{attribute 'GeneratedUsingTerminal: KL1382'}
{attribute addProperty BoxType "KL1382"}
{attribute addProperty Description ""}
{attribute addProperty Physics ""}
{attribute addProperty Id "Channel_1AT %I*Channel_22DCD6950Channel_2AT %I*Channel_22DCD6950"}
{attribute addProperty CRC "3041576269"}
{attribute addProperty Size "0"}
TYPE KL1382_B54AC54D :
STRUCT
	{attribute addProperty Name "Channel_1"}
	Channel_1 : Channel_22DCD695;
	{attribute addProperty Name "Channel_2"}
	Channel_2 : Channel_22DCD695;
END_STRUCT
END_TYPE

(* stored: Version 1.2.0.0, ProductVersion 3.1.4024.9
   DUT KL1382_B54AC54D: Id {fd5ecab8-9928-4b9e-936e-31967a66158a} *)
